TYPE "Positioning_EPOS_Machine_Alr"
VERSION : 0.1
// Block: Positioning_EPOS_Machine_Alr
   STRUCT
      S120_Fault : Bool;
      S120_ComErr : Bool;
      S120_WriteParErr : Bool;
      Ax_NotHomed : Bool;
      Ax_ErrSelMode : Bool;
      Ax_ErrOverride : Bool;
      Ax_InvalidTraversingBlockNr : Bool;
      HwLimitMinus : Bool;
      HwLimitPlus : Bool;
      BrakeTimeOut : Bool;
      Fan_M : MotorAlr;
   END_STRUCT;

END_TYPE
